// TIA Portal V17 export
// export: Created 2025-01-08T13:55:36.2416913Z, ExportSetting WithDefaults, DisplayName Totally Integrated Automation Portal, DisplayVersion V17, DisplayName TIA Portal Openness, DisplayVersion V17, DisplayName TIA Portal Version Control Interface, DisplayVersion V17, DisplayName SINAMICS Startdrive Advanced, DisplayVersion V17 Update2, DisplayName SINAMICS Startdrive G130, G150, S120, S150, SINAMICS MV, S210, DisplayVersion V17 Update2, DisplayName SINAMICS Startdrive G110M, G120, G120C, G120D, G120P, G115D, DisplayVersion V17 Update2, DisplayName STEP 7 Professional, DisplayVersion V17, DisplayName STEP 7 Safety, DisplayVersion V17, DisplayName WinCC Advanced, DisplayVersion V17
TYPE "DataFromHSM"
// stored: IsFailsafeCompliant false
   STRUCT
      Sts : Struct
         xStop : Bool;   // Setzt den Spender in Stopp
         xRun : Bool;   // Setzt den Spender in Run
         xService : Bool;
         xTeach : Bool;
         xFeed : Bool;
         xConfigurationSave : Bool;
         xConfigurationLoad : Bool;
         xReceiveConfiguration : Bool;
         xCParameterSend : Bool;   // Schreibt alle über Kparam Maske ausgewählten Kparameter auf die ACP
         xCParameterReceive : Bool;   // Schreibt alle über Kparam Maske ausgewählten Kparameter in den DB
         xMparameterSend : Bool;   // Schreibt alle über Mparam Maske ausgewählten Mparameter auf die ACP
         xMparameterReceive : Bool;   // Schreibt alle über Mparam Maske ausgewählten parameter auf die DB
         xReserved : Bool;
         xGetTime : Bool;
         xGet_MAC_FW_version : Bool;
         xStatusContinuouslyTransmitted : Bool;   // 1: Aktiviert die kontinuierliche übertragung des Control Registers
         xCommunicationMonitoring : Bool;
         "x AcknowledgeFaultFromExternal" : Bool;
         xBlockProductSensor : Bool;   // 1: Produktsensor ist nicht aktiv, d.h. es wird kein Etikettierimpuls ausgelöst
         xSplice_Start : Bool;
         xReserved_25 : Bool;
         xReserved_24 : Bool;
         xReserved_23 : Bool;
         xReserved_22 : Bool;
         xReserved_21 : Bool;
         xReserved_20 : Bool;
         xReserved_19 : Bool;
         xReserved_18 : Bool;
         xReserved_17 : Bool;
         xReserved_16 : Bool;
         xReserved_15 : Bool;
         xReserved_14 : Bool;
         xDeviceStatusOK : Bool;
         xDeviceStatusWarning : Bool;
         xDeviceStatusAlarm : Bool;
         xPauseRun : Bool;
         xPauseStandby : Bool;
         xPauseService : Bool;
         xLampAlarm : Bool;
         xLampOK : Bool;
         xLampWarning : Bool;
         "xIO-Warning" : Bool;
         "xIO-Ready" : Bool;
         "xIO-Sync" : Bool;
         xSync2 : Bool;
         xSync3 : Bool;
         xLabelSensor : Bool;
         xProductSensorPolarity : Bool;
         xLowLabelSensor : Bool;
         xWebBreakSensor : Bool;
         xExternalStart : Bool;
         xSpliceActive : Bool;
         xReserved_12 : Bool;
         xReserved_11 : Bool;
         xReserved_10 : Bool;
         xReserved_09 : Bool;
         xReserved_08 : Bool;
         xReserved_07 : Bool;
         xReserved_06 : Bool;
         xReserved_05 : Bool;
         xReserved_04 : Bool;
         xReserved_03 : Bool;
         xReserved_02 : Bool;
         xReserved_01 : Bool;
         iLabelCounter : Int;
         iCounterRemaining : Int;
         iMcurr : Int;   // Status- Mittlerer Motorstrom in %
         wExtEncoder : Word;   // Status- Zählerwert des Ext. Encoders
         wErrorCode : Word;   // Fehlerwert
         wWarnNr : Word;   // Warnungscodes
         iReserved_W1 : Int;
         iReserved_W2 : Int;
         iReserved_W3 : Int;
         iReserved_W4 : Int;
         iReserved_W5 : Int;
         iReserved_W6 : Int;
      END_STRUCT;
      Cfg : Struct
         iLabellingSpeed : Int;   // in 1/10 m/min
         iTriggerDelay : Int;   // in 1/10 mm
         iLabelPosition : Int;   // in 1/10 mm
         iLabelLenght : Int;   // in mm
         iLabelGap : Int;   // in 1/10 mm
         iLabelsBurst : Int;   // 1=Aus, 2=zweimal … (mehrere Etiketten mit einem Triggerimpuls)
         iDistanceBetweenLabels : Int;   // in 1/10 mm (Abstand zwischen den Etiketten wenn mehrere pro Trigger)
         iMaxNumberOfLabelsToSkip : Int;   // 0 - n
         iTriggerBlank : Int;   // in mm
         iAccelerationRamp : Int;   // in 1/10 mm
         iSpeedInternalEncoder : Int;   // 0 = Intern, 1 = Drehgeber
         iStopRamp : Int;   // in % (Verhältnis zur Startrampe)
         iSyncOutputDelay : Int;   // in 1/10 mm
         iSyncOutputLength : Int;   // in 1/10 mm
         iSyncOutputDelay2 : Int;   // in 1/10 mm
         iSyncOutputLenght_2 : Int;   // in 1/10 mm
         iSyncOutputDelay_3 : Int;   // in 1/10 mm
         iSyncOutputLenght_3 : Int;   // in 1/10 mm
         iPreFeed : Int;   // in 1/10 mm
         iConveyorSpeed_1 : Int;
         iConveyorSpeed_2 : Int;
         iReserved_11 : Int;
         iReserved_10 : Int;
         iReserved_09 : Int;
         iReserved_08 : Int;
         iReserved_07 : Int;
         iReserved_06 : Int;
         iReserved_05 : Int;
         iReserved_04 : Int;
         iReserved_03 : Int;
         iReserved_02 : Int;
         iReserved_01 : Int;
      END_STRUCT;
      M_Par : Struct
         iSpeedInternalEncoder : Int;   // 0 = Fixed internally, 1 = Encoder fixed, 2 = Value from configuration
         iEncoderMMPerRevolution : Int;   // in 1/10 mm
         iEncoderPulsesPerRevolution : Int;   // in Pulse
         iMaximumSpeed : Int;   // in 1/10 m/min
         iInstallationMode : Int;   // 0 = normal, 1 = feed also via start button, 2 = feed with fixed length via start button, 3 = feed always with fixed length
         iLabelLengthInMMPerMotorRevolution : Int;   // in 1/100 mm
         iDistanceGapSensorToDispensingEdge : Int;   // in 1/10 mm
         iProductSensorPolarity : Int;   // 0 = NPN, 1 = NPN inverted, 2 = PNP inverted, 3 = PNP
         iSkipMode_1 : Int;   // 0 = value from configuration, 1 = value from machine parameters, 2 = end detect
         iMaxLabelSkip : Int;   // 0 - n
         iAccelerationMode : Int;   // 0 = value from configuration, 1 = value from machine parameters
         iAcceleration : Int;   // in 1/10 mm
         iGapSensor : Int;   // 0 = leading edge, 1 = trailing edge label
         iMaxCalibrationLength : Int;   // in 1/10mm
         iDecelarationMode : Int;   // 0 = value from configuration, 1 = value from machine parameters
         iDecelaration : Int;   // in % (of acceleration distance)
         iExernalStart : Int;   // 0 = off 1 = edge controlled 2 = pulse controlled
         iLowLabelInput : Int;   // 0= Off 1=On
         iBeltInput_1 : Int;   // 0= Off 1=On
         iSyncParameter_1 : Int;   // 0 = value from configuration, 1 = value from machine parameters
         iSyncOutputDelay : Int;   // in 1/10mm
         iSyncOutputLength : Int;   // in 1/10mm
         iZeroDownTimeMode_1 : Int;   // 0 = off 1 = master 2 = slave
         iZeroDownTimeSensorDistance : Int;   // in mm
         iLabelLengthInCaseOfErrorOnLowLabelSensor : Int;   // in m
         iLowLabelSensorPolarity : Int;   // 2 = PNP inverted 3 = PNP
         iWebBreakSensorPolarity : Int;   // 2 = PNP inverted 3 = PNP
         iWarningOutputPolarity_1 : Int;   // 2 = PNP inverted 3 = PNP
         iSync2Parameter_1 : Int;   // 0 = value from configuration, 1 = value from machine parameters
         iSync2OutputDelay_1 : Int;   // in 1/10mm
         iSync2OutputPulseLength_1 : Int;   // in 1/10mm
         iSync3Parameter_1 : Int;   // 0 = value from configuration, 1 = value from machine parameters
         iSync3OutputDelay_1 : Int;   // in 1/10mm
         iSync3OutputPulseLength_1 : Int;   // in 1/10mm
         iTeachTolerance : Int;   // in 1/100mm
         iSynch1Mode_1 : Int;   // 0 = production sensor 1 = trigger sensor 2 = reserve 3 = end of dispensing
         iSynch2Mode_1 : Int;   // 0 = production sensor 1 = trigger sensor 2 = reserve 3 = end of dispensing
         iSynch3Mode_1 : Int;   // 0 = production sensor 1 = trigger sensor 2 = reserve 3 = end of dispensing
         iOvercurrentCorrection : Int;   // in %
         iServiceFeedSpeed : Int;   // in 1/10 m/min
         iPreDispensingMode : Int;   // 0 = value from configuration, 1 = value from machine parameters
         iPreDispensingLength : Int;   // in 1/10 mm
         iLabelSensorWindowPreDispensingPath : Int;   // in 1/10 mm
         iLabelSensorCount : Int;
         "iSPS-Mode_1" : Int;   // 0 = Off 1 = S7 communication / 0= Off 1= S7-communication, 2 = S7-communication double size
         iZdtWin_1 : Int;   // Zero down time window mm / Zero Down Time Window mm
         iDistRes_1 : Int;   // Resolution label spacing
         "iSPS-DB-NoCtrl_1" : Int;   // SPS-DB-Nr Control (SPS->ACP) / Data block for PLC communication
         "iSPS-DB-NoStat_1" : Int;   // SPS-DB-Nr Status (ACP->SPS) / Data block for PLC communication
         iSignalFormat_1 : Int;   // Status-Server: Signalform / Is relevant for the WEBER-TOOL
         iLowLabDiam_1 : Int;   // Roll diameter for LowLabel in 1/10 mm / Roll diameter for LowLab in 1/10 mm
         iCoreDiameter_1 : Int;   // Core diameter in 1/10 mm
         iWebBreakRest_1 : Int;   // Rest after WebBreak in mm
         iLeverSetup_1 : Int;   // Do not use here / To the TEACH of the dancer position
         iLeverMinPos_1 : Int;   // Analog value angle sensor unwinder dancer Min.Pos.
         iLeverMaxPos_1 : Int;   // Analog value angle sensor unwinder dancer Max.Pos.
         "iUW-BufLength_1" : Int;   // Label path in mm between dancers min / max
         iTwinLabelMd_1 : Int;   // Double Label Mode / Double Label mode
         iLabelQueTolerans : Int;   // Setting the tolerance "Number of labels between peel bar and label sensor".
         iResetEvents : Int;   // Reset the operating data EV#007 „Number of all spent labels“ or EV#008 „Display of label roll dispensed“. 0 = off, 1 = reset EV#007 Label feeds, 2 = reset EV#008 Label meters.
         iMaintenanceDistanceKm : Int;   // Setting the maintenance interval depending on the the label roll length. [km]
         iMaintenanceDays : Int;   // Setting the maintenance interval depending on the operation time. [days]
         iProductSensorMode : Int;   // Defines the linkage of the product sensors 1 and 2 with respect to the trigger signal. 0 = Off, 1 = AND Operation (both sensors must recieve a signal), 2 = OR operation (only one sensor have to recieve a signal)
         iRewinderDiameterWarning : Int;   // Defines the diameter of the carrier web, after which a pre-warning for the rewinder is avti-vated. The following message appears "Rewinder almost full".
         arrayFirmwareVersion_1 : Array[0..19] of Char;   // Defines the diameter of the carrier web, after which the labeler stops. The following mes-sage appears "Rewinder full".
         "arrayCfg_MAC-Adress_1" : Array[0..19] of Char;   // Defines the value for the motor current, after which the following message appears "Load approaching the upper limit".
         iRewinderDiameterFull : Int;   // Parameter for activating contour mode. When the parameter is activated, the two parameters "Start contour" and "Stop contour" are displayed in the configuration menu. At the same time, the "Ramp" parameter is ignored.
         iMotorLoadLimit : Int;   // Determines the number of encoder pulses per millimeter of label path and synchronizes an optional printer at the AUX socket.
         iCountorRamp : Int;   // This Parameter is used to set the communication with different PLC versions.
         iEncoderOutPulsMM : Int;   // This parameter is used to set the distance (duration) in splice mode. The label web is ad-vanced with the reduced speed specified in parameter 071. 0 - 9999. Adjusting the value in [mm]
         iSPS_RackAndSlot : Int;   // This parameter is only used if parameter 070 is active. It is used to reduce reduce the speed in the slice mode and is calculated on the basis of the current speed. 10 - 100. Adjusting the value in [%]
         iSpliceDistance : Int;   // This parameter is only used for alternating operation and defines the transfer reserve that is still to be dispensed in alternating operation. Must be less than or equal to Par.25 RestLowLabel. 0.0 – 90.0. Adjusting the value in [m]
         iSpliceSpeedReduction : Int;   // Offset setting for operation with rotary encoder. The feed rate of the dispenser is factor Par.73 x encoder speed. 20.0 - 500.0. Adjusting the value in [%].
         iDownstream : Int := 20;   // Setting of the start ramp setting in m/s2. If the value is 0, the ramp length is used to calcu-late the acceleration. The stop ramp is set exactly as before via the ratio to the start ramp. 0.0 - 90.0. In [m/s2]
         iSpeedFactor : Int := 1000;   // Setting of a speed offset in 1/10 m/min. Only applies to the internal speed. Parameter 073 can be used in encoder mode. -20.0 - 20.0. in [%]
         iAcceleration_1 : Int := 0;   // Determines whether the material transport error "Materialtransportoffen" is to be output. The signal for the error must be applied to X22.4. 0 = Off. 1 = Error at 24V. 2 = Error at 0V.
         iSpeedOffset : Int := 0;   // Offset setting of the encoder speed for the internal calculation of Alpha HSM, e.g. for win-ding tape operation and ZDT application. Alpha HSM must calculate with baseband speed for the function of the ZDT, but dispenses with encoder speed from the winding belt. 20.0 - 500.0. In [%]
         iMaterialTransportErrorMode : Int := 0;   // Determines whether the material transport error "Materialtransportoffen" is to be output. The signal for the error must be applied to X22.4. 0 = Off. 1 = Error at 24V. 2 = Error at 0V.
         iEncoderFactor : Int := 1000;   // Offset setting of the encoder speed for the internal calculation of Alpha HSM, e.g. for win-ding tape operation and ZDT application. Alpha HSM must calculate with baseband speed for the function of the ZDT, but dispenses with encoder speed from the winding belt. 20.0 - 500.0. In [%]
         iReserve_1 : Int;
         iReserve_2 : Int;
         iReserve_3 : Int;
         iReserve_4 : Int;
         iReserve_5 : Int;
         iReserve_6 : Int;
         iReserve_7 : Int;
         iReserve_8 : Int;
         iReserve_9 : Int;
         iReserve_10 : Int;
         iReserve_11 : Int;
         iReserve_12 : Int;
         iReserve_13 : Int;
         iReserve_14 : Int;
         iReserve_15 : Int;
         iReserve_16 : Int;
         iReserve_17 : Int;
         iReserve_18 : Int;
         iReserve_19 : Int;
         iReserve_20 : Int;
         iReserve_21 : Int;
         iReserve_22 : Int;
         iReserve_23 : Int;
         iReserve_24 : Int;
         iReserve_25 : Int;
         iReserve_26 : Int;
         iReserve_27 : Int;
         iReserve_28 : Int;
         iReserve_29 : Int;
         iReserve_30 : Int;
         iReserve_31 : Int;
         iReserve_32 : Int;
         iReserve_33 : Int;
         iReserve_34 : Int;
         iReserve_35 : Int;
         iReserve_36 : Int;
         iReserve_37 : Int;
         iReserve_38 : Int;
         iReserve_39 : Int;
         iReserve_40 : Int;
         iReserve_41 : Int;
         iReserve_42 : Int;
         iReserve_43 : Int;
         iReserve_44 : Int;
         iReserve_45 : Int;
         iReserve_46 : Int;
         iReserve_47 : Int;
         iReserve_48 : Int;
         iReserve_49 : Int;
         iReserve_50 : Int;
         iReserve_51 : Int;
      END_STRUCT;
   END_STRUCT;
END_TYPE
